# EPICS StreamDevice protocol: laser-ioc/laserApp/Db/laser.proto
#setPWM {
#    out "PWM_SET %f";
#}

#enablePWM {
#    out "PWM_ENABLE %d";
#}

Terminator = LF;

setPWM {
    out "PWM_SET %f";
    #in "OK";
}

enablePWM {
    out "PWM_ENABLE %d";
    #in "OK";
}
